RoboDK station: Celda Robotica.rdk

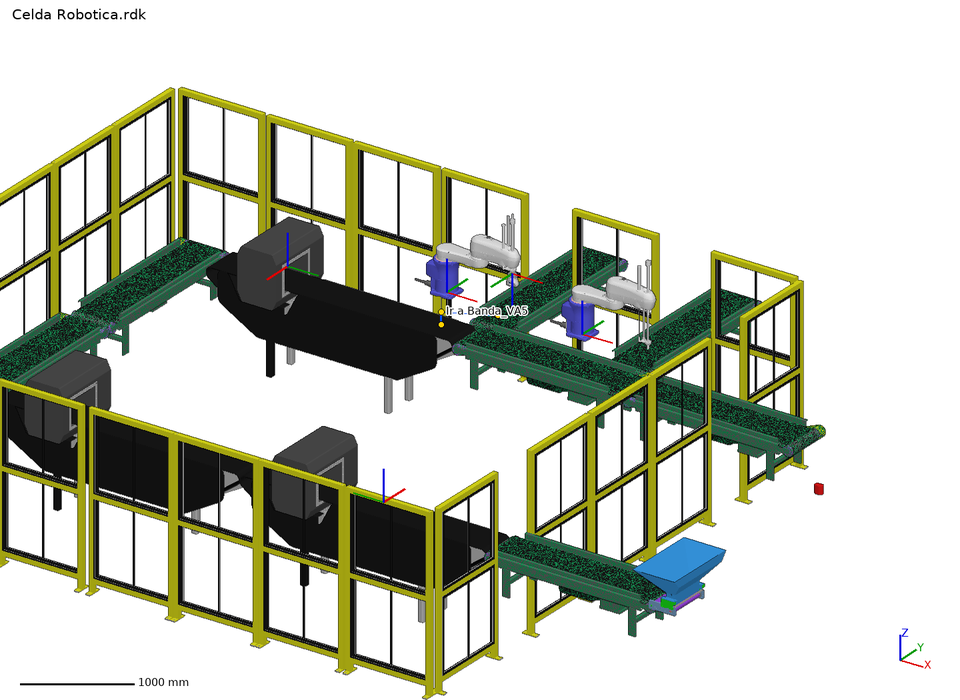
[picture v0: the station drawn from its stored meshes, robots at their saved joint values, targets as dots, program paths as lines]
Station Celda Robotica (saved by RoboDK 5.2.5). Poses are relative to the parent item; angles as X-Y-Z fixed-axis rotations.
  - frame Robot 1 at (-1950, 3750, 0) mm
    - robot Denso HM-4A73 1 (model Denso HM-4A73): 4 axes, payload 20 kg, reach 700 mm, repeatability 0.022 mm, weight 56 kg
        modified DH rows (alpha deg, a mm, theta deg, d mm): 0, 0, 0, 0; 0, 350, 0, 0; 0, 350, 0, 46 linear; 180, 0, 0, 0
        joint limits [-165, -147, 130, -360] to [0, 147, 300, 360]; home [0, 0, 300, 0]; saved at [0, 0, 300, 0]
      - frame Schunk_Gripper Base at (0, 0, -34) mm
        - robot Schunk_Gripper 1: 1 axes
            joint limits [0] to [40]; home [0]; saved at [40]
          - tool Schunk_Gripper, TCP at (0, 0, 200) mm, size 113.9 x 87 x 115.9 mm, geometry from Shunk_Gripper.sld
          - tool Schunk_Finger_1, TCP at (0, 0, 200) mm, size 58.3 x 33.9 x 89.4 mm, geometry from Shunk_Finger_1.sld
          - tool Schunk_Finger_2, TCP at (0, 0, 200) mm, size 58.3 x 34 x 89.4 mm, geometry from Shunk_Finger_2.sld
        - target Open (joint target) at (0, 0, 350) mm; joints [40] of Schunk_Gripper 1
        - target Close (joint target) at (0, 0, 350) mm; joints [0, 0, 0, 0] of Schunk_Gripper 1
        - target Tomar (joint target) at (0, 0, 350) mm; joints [28.44] of Schunk_Gripper 1
      - tool Schunk_TCP, TCP at (0, 0, 200) mm
    - target Ir a Banda_VA5 (Cartesian target) at (354.74, -592.38, 146) mm, rotated rx 180 ry 0 rz -95.82 deg; joints [-49.62, -18.93, 300, 27.27] of Denso HM-4A73 1
    - target Ir a Banda_Selec6 (Cartesian target) at (658.71, -159.66, 24.85) mm, rotated rx 180 ry 0 rz 0.85 deg; joints [-28.1, 28.95, 178.85, 0] of Denso HM-4A73 1
  - frame Robot 2 at (-500, 3750, 0) mm
    - robot Denso HM-4A73 2 (model Denso HM-4A73): 4 axes, payload 20 kg, reach 700 mm, repeatability 0.022 mm, weight 56 kg
        modified DH rows (alpha deg, a mm, theta deg, d mm): 0, 0, 0, 0; 0, 350, 0, 0; 0, 350, 0, 46 linear; 180, 0, 0, 0
        joint limits [-165, -147, 0, -360] to [165, 147, 300, 360]; home [0, 0, 0, 0]; saved at [0.018, -0.037, 0, -0.018]
  - frame Celda Robotica at (0, 0, 0) mm, rotated rx 0 ry 0 rz 90 deg
    - object Tolva_Distribucion_1 at (0, 0, 0) mm, size 480.2 x 432.5 x 787.5 mm, geometry from CONVEYOR WITH HOPPER.STEP
    - object Banda_Suministro_1 at (0, 0, 0) mm, size 527 x 431.8 x 1828.4 mm, geometry from Horizontal belt conveyor.step
    - object Banda_Filtrado_2 at (0, 0, 0) mm, size 2639.7 x 1260 x 880.5 mm, geometry from _ASSY, METAL DETECTOR 1069.STL
    - object Banda_Enjuague_3 at (0, 0, 0) mm, size 2639.7 x 1260 x 880.5 mm, geometry from _ASSY, METAL DETECTOR 1069.STL
    - object Banda_Escurrido_4a at (0, 0, 0) mm, size 527 x 431.8 x 1828.4 mm, geometry from Horizontal belt conveyor.step
    - object Banda_Escurrido_4b at (0, 0, 0) mm, size 527 x 431.8 x 1828.4 mm, geometry from Horizontal belt conveyor.step
    - object Banda_Visio_Artificial_5 at (0, 0, 0) mm, size 2639.7 x 1260 x 880.5 mm, geometry from _ASSY, METAL DETECTOR 1069.STL
    - object Banda_Seleccion_6 at (0, 0, 0) mm, size 527 x 431.8 x 1828.4 mm, geometry from Horizontal belt conveyor.step
    - object Banda_Seleccion_7 at (0, 0, 0) mm, size 527 x 431.8 x 1828.4 mm, geometry from Horizontal belt conveyor.step
    - object Banda_Merma_8a at (0, 0, 0) mm, size 527 x 431.8 x 1828.4 mm, geometry from Horizontal belt conveyor.step
    - object Banda_Merma_8b at (0, 0, 0) mm, size 527 x 431.8 x 1828.4 mm, geometry from Horizontal belt conveyor.step
    - object Barda_Seguridad_9 at (0, 0, 0) mm, size 900 x 1800 x 150 mm, geometry from Security_frame.STEP
      - object BS_9a at (0, 0, 0) mm, size 900 x 1800 x 150 mm, geometry from Security_frame.STEP
      - object BS_9b at (0, 0, 0) mm, size 900 x 1800 x 150 mm, geometry from Security_frame.STEP
      - object BS_9c at (0, 0, 0) mm, size 900 x 1800 x 150 mm, geometry from Security_frame.STEP
      - object BS_9d at (0, 0, 0) mm, size 900 x 1800 x 150 mm, geometry from Security_frame.STEP
      - object BS_9e at (0, 0, 0) mm, size 900 x 1800 x 150 mm, geometry from Security_frame.STEP
      - object BS_9f at (0, 0, 0) mm, size 900 x 1800 x 150 mm, geometry from Security_frame.STEP
      - object BS_9g at (0, 0, 0) mm, size 900 x 1800 x 150 mm, geometry from Security_frame.STEP
      - object BS_9h at (0, 0, 0) mm, size 900 x 1800 x 150 mm, geometry from Security_frame.STEP
      - object BS_9i at (0, 0, 0) mm, size 900 x 1800 x 150 mm, geometry from Security_frame.STEP
      - object BS_9j at (0, 0, 0) mm, size 900 x 1800 x 150 mm, geometry from Security_frame.STEP
      - object BS_9k at (0, 0, 0) mm, size 900 x 1800 x 150 mm, geometry from Security_frame.STEP
      - object BS_9l at (0, 0, 0) mm, size 900 x 1800 x 150 mm, geometry from Security_frame.STEP
      - object BS_9m at (0, 0, 0) mm, size 900 x 1800 x 150 mm, geometry from Security_frame.STEP
      - object BS_9n at (0, 0, 0) mm, size 900 x 1800 x 150 mm, geometry from Security_frame.STEP
      - object BS_9o at (0, 0, 0) mm, size 900 x 1800 x 150 mm, geometry from Security_frame.STEP
      - object BS_9p at (0, 0, 0) mm, size 900 x 1800 x 150 mm, geometry from Security_frame.STEP
      - object BS_9q at (0, 0, 0) mm, size 900 x 1800 x 150 mm, geometry from Security_frame.STEP
      - object BS_9r at (0, 0, 0) mm, size 900 x 1800 x 150 mm, geometry from Security_frame.STEP
      - object BS_9s at (0, 0, 0) mm, size 900 x 1800 x 150 mm, geometry from Security_frame.STEP
      - object BS_9t at (0, 0, 0) mm, size 900 x 1800 x 150 mm, geometry from Security_frame.STEP
      - object BS_9u at (0, 0, 0) mm, size 900 x 1800 x 150 mm, geometry from Security_frame.STEP
      - object BS_9v at (0, 0, 0) mm, size 900 x 1800 x 150 mm, geometry from Security_frame.STEP
      - object BS_9w at (0, 0, 0) mm, size 900 x 1800 x 150 mm, geometry from Security_frame.STEP
  - program Robot1_CloseGripper (3 instructions, listed below)
  - program Robot1_OpenGripper (1 instructions, listed below)
  - program Robot1_Tomar (1 instructions, listed below)
  - program Robot1_PickChile (11 instructions, listed below)
  - frame ConveyorReference at (-3387.94, 3378.09, 0) mm, rotated rx 0 ry 0 rz -89.76 deg
    - object Conveyor at (0, 300, -50) mm, size 597 x 2090.8 x 107.2 mm
      - Python program RunConveyor (listed below)
      - Python program SimulateGripper (listed below)
      - object Part 7 at (225.23, 5502.13, -410) mm, size 60 x 60 x 80 mm
      - object Part 2 at (225.26, 5504.63, -410) mm, size 60 x 60 x 80 mm
      - object Part 3 at (225.26, 5512.28, -410) mm, size 60 x 60 x 80 mm
      - object Part 4 at (225.26, 5508.44, -410) mm, size 60 x 60 x 80 mm
      - object Part 8 at (225.26, 5522.21, -410) mm, rotated rx 0 ry 0.16 rz 0 deg, size 60 x 60 x 80 mm
      - object Part 1 at (225.26, 5504.71, -410) mm, size 60 x 60 x 80 mm
      - object Part 5 at (225.26, 5529.4, -410) mm, size 60 x 60 x 80 mm
      - object Part 6 at (225.26, 5518.61, -410) mm, size 60 x 60 x 80 mm
    - target Get Conveyor (joint target) at (227.58, 1791.75, 21.09) mm, rotated rx 180 ry 0 rz -0.61 deg; joints [-49.427, -19.281, 175.095, 21.662] of Denso HM-4A73 1
  - Python program WaitForPart (listed below)
  - program Principal (11 instructions, listed below)
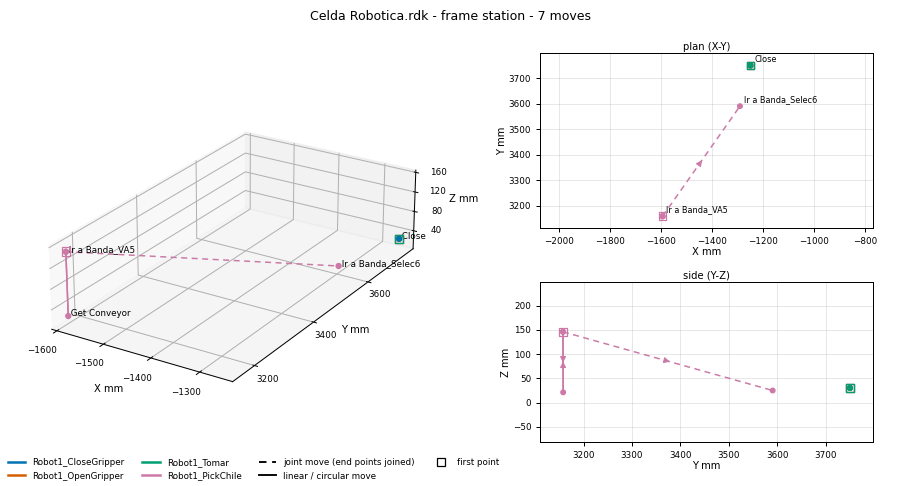
[picture p0: tool path of Celda Robotica.rdk in frame station, 7 of 7 moves have a stored position in this frame; points joined in program order, loops and branches not executed]

--- program Robot1_CloseGripper (robot Schunk_Gripper 1) ---
  Est. Ref.: Schunk_Gripper Base
  Est. herr: Schunk_Gripper
  MoveJ (Close)

--- program Robot1_OpenGripper (robot Schunk_Gripper 1) ---
  MoveJ (Open)

--- program Robot1_Tomar (robot Schunk_Gripper 1) ---
  MoveJ (Tomar)

--- program Robot1_PickChile (robot Denso HM-4A73 1) ---
  Est. Ref.: Robot 1
  Est. herr: Schunk_TCP
  MoveJ (Ir a Banda_VA5)
  MoveL (Target 1) -> target Get Conveyor
  Llamar WaitForPart
  Llamar Robot1_Tomar
  Adjuntar a Schunk_Gripper
  MoveL (Ir a Banda_VA5)
  MoveJ (Ir a Banda_Selec6)
  Llamar Robot1_OpenGripper
  Separar de Schunk_Gripper

--- Python program RunConveyor ---
# Type help("robolink") or help("robodk") for more information
# Press F5 to run the script
# Note: you do not need to keep a copy of this file, your python script is saved with the station
from robolink import *    # API to communicate with RoboDK
from robodk import *      # basic matrix operations
RDK = Robolink()

# This script simulates a conveyor belt
CONVEYOR_NAME = 'Conveyor'
PICKABLE_OBJECTS_KEYWORD = 'Part'

# Speed of movement in MM/S with respect to the conveyor coordinates:
MOVE_SPEED_MMS = [0,10,0]
REFRESH_RATE = 0.005

# Define workspace of the conveyor to pick the objects:
CONV_SZ_X_MIN = 0
CONV_SZ_X_MAX = 440
CONV_SZ_Y_MIN = 0
CONV_SZ_Y_MAX = 5800
CONV_SZ_Z_MIN = -200
CONV_SZ_Z_MAX = +500

# Move objects that reached the end of the conveyor and were not picked:
FALLEN_OBJECTS = [0,0,-500]

# Get the conveyor item and reference for work space:
conv = RDK.Item(CONVEYOR_NAME)
conv_reference = conv.Parent()
poseconv = conv_reference.PoseAbs()

# One second in real life means 1 second of simulation. The simulation speed is taken from the station
SIMULATION_SPEED = 1

def is_inside_conveyor(pose):
    """Checks if a pose is inside the conveyor workspace"""
    pos = pose.Pos()
    if pos[0] > CONV_SZ_X_MIN and pos[0] < CONV_SZ_X_MAX and pos[1] > CONV_SZ_Y_MIN and pos[1] < CONV_SZ_Y_MAX and pos[2] > CONV_SZ_Z_MIN and pos[2] < CONV_SZ_Z_MAX:
        return True
    return False

def conveyor_move_object(pose, delta_time):
    """Moves the object pose through the conveyor depending on the time and speed"""
    delta_mm = mult3(MOVE_SPEED_MMS, delta_time)
    newpose = transl(delta_mm)*pose
    return newpose

# Get all objects (string list)
all_objects = RDK.ItemList(ITEM_TYPE_OBJECT, True)

# Convert object list into item pointers (faster)
# Also filter the list to take into account pickable objects only
objects = []
objects_name = []
objects_active = []
for i in range(len(all_objects)):
    if all_objects[i].count(PICKABLE_OBJECTS_KEYWORD) > 0:
        objects.append(RDK.Item(all_objects[i]))
        objects_name.append(all_objects[i])
        objects_active.append(False)

# The number of objects that can go in the conveyor
nobjects = len(objects)


# Infinite loop to simulate the conveyor behavior
current_time = 0
tic()
time_last = toc()
while True:
    # First: Look for objects that are not in the conveyor but are in the conveyor workspace
    for i in range(nobjects):
        obj_i = objects[i]

        # Skip if the object is already in the conveyor
        if objects_active[i]:
            continue

        # Check if the object has already been taken by a tool. If so, do not take it in the conveyor
        if obj_i.Parent().Type() == ITEM_TYPE_TOOL:
            continue

        # Check if the object is within the conveyor work area
        posei = obj_i.PoseAbs()
        poseirel = invH(poseconv)*posei
        if is_inside_conveyor(poseirel):
            # take the object
            obj_i.setParentStatic(conv)
            print('Adding object %s to the conveyor' % objects_name[i])
            objects_active[i] = True

    # Second step: Update the position of every object in the conveyor
    SIMULATION_SPEED = RDK.SimulationSpeed()
    time_current = toc()
    time_delta = time_current - time_last
    time_last = time_current
    current_time = current_time + time_delta*SIMULATION_SPEED

    # Make a list of objects with their matching positions to update
    obj_items = []
    obj_poses_abs = []
    for i in range(nobjects):
        obj_i = objects[i]

        # Check if the object has been picked from the conveyor
        if objects_active[i] and not obj_i.Parent().equals(conv):
            objects_active[i] = False
            print('Object %s was picked from the conveyor' % objects_name[i])
            continue

        # Skip update for objects that are not in the conveyor
        if not objects_active[i]:
            continue

        # Update the position of the object
        posei = invH(poseconv)*obj_i.PoseAbs()
        newposei = conveyor_move_object(posei, time_delta*SIMULATION_SPEED)
        if not is_inside_conveyor(newposei):
            print('Warning!! Object %s fell from the conveyor at %.1f seconds after simulation started' % (objects_name[i], current_time))
            #raise Exception('Object %s was not picked from the conveyor!' % objects_name[i])
            newposei = transl(FALLEN_OBJECTS)*newposei
            objects_active[i] = False

        #obj_i.setPose(newposei) # this will provoke a refresh (can be slow)
        obj_items.append(obj_i)
        obj_poses_abs.append(poseconv*newposei)

    # Update the object positions
    RDK.setPosesAbs(obj_items, obj_poses_abs)

    # Take a break...
    pause(REFRESH_RATE)

--- Python program SimulateGripper ---
# Type help("robolink") or help("robodk") for more information
# Press F5 to run the script
# Note: you do not need to keep a copy of this file, your python script is saved with the station
from robolink import *    # API to communicate with RoboDK
from robodk import *      # basic matrix operations
RDK = Robolink()

# This file allows simulating the opening and closing of grippers.
# Two models of the gripper per robot are required: one opened and one closed.
# The opened model of the gripper should have the keyword "Opened"
# The closed model of the gripper should have the keyword "Closed"
# Simply place this file in the station and leave it running to
# make it work

OPENED_KEYWORD = 'Opened'
CLOSED_KEYWORD = 'Closed'
UPDATE_FREQUENCY = 0.01

# Loop forever
print('Starting infinite loop to simulate open/close of tools')
while True:
    # First step: get a list of tool pairs (open, closed) per robot
    Tool_Pairs = []
    # get all the robot names (strings)
    all_robots = RDK.ItemList(ITEM_TYPE_ROBOT)
    for i in range(len(all_robots)):
        roboti = RDK.Item(all_robots[i])
        roboti_name = roboti.Name()
        # get the tools of each robot
        roboti_tools = roboti.Childs()
        opened = None
        closed = None
        # store the opened model and closed model of each gripper
        for t in range(len(roboti_tools)):
            tnamei = roboti_tools[t].Name()
            if not isinstance(opened,Item) and tnamei.count(OPENED_KEYWORD) > 0:
                opened = roboti_tools[t]
                print('Using %s from robot %s as gripper opened' % (tnamei, roboti_name))
            elif not isinstance(closed,Item) and tnamei.count(CLOSED_KEYWORD) > 0:
                closed = roboti_tools[t]
                print('Using %s from robot %s as gripper closed' % (tnamei, roboti_name))

            if isinstance(opened, Item) and isinstance(closed, Item):
                # Stop if we have an open state and a closed state per robot
                break;
        Tool_Pairs.append([opened, closed])

    # We may find as many pairs of tools as robots are available in the station
    nTool_Pairs = len(Tool_Pairs)
    while True:
        #try:
            # Iterate through all tool pairs and detect the presence of objects
            for i in range(nTool_Pairs):
                opened = Tool_Pairs[i][0]
                closed = Tool_Pairs[i][1]
                open_valid = isinstance(opened,Item)
                close_valid = isinstance(closed,Item)
                tool_is_open = True

                # Check if the tool holds one or more objects:
                if (open_valid and len(opened.Childs()) > 0) or (close_valid and len(closed.Childs()) > 0):
                    tool_is_open = False

                # Update the visibility of the tools
                if open_valid:
                    opened.setVisible(tool_is_open)
                if close_valid:
                    closed.setVisible(not tool_is_open)

            # Take a pause...
            pause(UPDATE_FREQUENCY)

        #except:
            #print('An item was deleted. Remaking tool list')
            #break

--- Python program WaitForPart ---
# Type help("robolink") or help("robodk") for more information
# Press F5 to run the script
# Note: you do not need to keep a copy of this file, your python script is saved with the station
from robolink import *    # API to communicate with RoboDK
from robodk import *      # basic matrix operations
RDK = Robolink()

# RDK.ShowMessage('Hola', popup=False)

# This script allows to simulate a laser sensor
# that detect the presence of a part in a plane,
# such as a part crossing a laser sensor in a
# conveyor belt

# The script finishes once a part has been detected
# so it works like a WAIT UNTIL function.

# Use a target from the station as a reference plane:
TARGET_NAME = 'Get Conveyor'
LASER_PLANE = [-1,0,0] # normal of the plane

# Activate within this tolerance
TOLERANCE_CHECK_MM = 20

# Look for parts with the keyword "Part"
PICKABLE_OBJECTS_KEYWORD = 'Part'

# Update status every 1 ms
RECHECK_PERIOD = 0.001

# Get the target and the detection plane
target = RDK.Item(TARGET_NAME)
targetpose = target.PoseAbs()
DETECT_PLANE_POINT = targetpose.Pos()
DETECT_PLANE_VECTOR = LASER_PLANE

# Define a function to detect a target
def part_detected(pos):
    """Check if a part is in the detection area (proximity of a point to a plane)"""
    pos_proj = proj_pt_2_plane(pos, DETECT_PLANE_POINT, DETECT_PLANE_VECTOR)
    distance2plane = norm(subs3(pos,pos_proj))
    if distance2plane < TOLERANCE_CHECK_MM:
        return True
    return False

# Get all object names
all_objects = RDK.ItemList(ITEM_TYPE_OBJECT, True)

# Get object items in a list (faster) and filter by keyword
check_objects = []
check_objects_names = []
for i in range(len(all_objects)):
    if all_objects[i].count(PICKABLE_OBJECTS_KEYWORD) > 0:
        check_objects_names.append(all_objects[i])
        check_objects.append(RDK.Item(all_objects[i]))

# Make sure that there are part that we are expecting
nCheck_objects = len(check_objects)
if nCheck_objects == 0:
    raise Exception('No parts to check for. The keyword is %s.' % PICKABLE_OBJECTS_KEYWORD)

# Loop forever until a part is detected by the sensor
part_available = False;
while not part_available:
    for i in range(nCheck_objects):
        if part_detected(check_objects[i].PoseAbs().Pos()):
            print('Part detected: %s' % check_objects_names[i])
            part_available = True
            break

    # Wait some time...
    pause(RECHECK_PERIOD)

print('Procedure finished')

--- program Principal (robot Denso HM-4A73 1) ---
  Llamar Robot1_OpenGripper
  Reemplazar objetos
  Ejecutar RunConveyor
  Llamar Robot1_PickChile
  Llamar Robot1_PickChile
  Llamar Robot1_PickChile
  Llamar Robot1_PickChile
  Llamar Robot1_PickChile
  Llamar Robot1_PickChile
  Llamar Robot1_PickChile
  Llamar Robot1_PickChile
